Fanuc KAREL source: kt00065.KL

-- PROVISIONAL review KL for V1013-1; original PC SHA256 da25708d8096a6e884967dbde137e86de862aeaaf0db347661e8ac84f2bec27e
-- Incomplete behavior may be omitted. Consult companion uncertainty JSON. Do not deploy.
PROGRAM KT00065
%NOLOCKGROUP
VAR
  I1 : INTEGER
  I2 : INTEGER
  OUT : INTEGER
BEGIN
  -- UNRESOLVED_PC offsets 5-16; opcodes 2E,23
  -- UNRESOLVED_PC offsets 21-32; opcodes 2E,23
  -- UNRESOLVED_PC offsets 37-48; opcodes 2E,23
  -- UNRESOLVED_PC offsets 53-64; opcodes 2E,23
  -- UNRESOLVED_PC offsets 69-88; opcodes 21,21,54,23
  -- UNRESOLVED_PC offsets 93-97; opcodes 7F
END KT00065
